(* PLC project copie_batch, Dassault Systèmes ControlBuild 2024x Refresh1 *)
(* stored: creationDateTime 2024-04-12T14:05:58-01:00 *)

PROGRAM gene_panel
  VAR_OUTPUT
    acknowledgePB : BOOL := false;
  END_VAR
  VAR_OUTPUT
    powerUp : BOOL := false;
    emergencyStop : BOOL := false;
    manualSwitch : BOOL := false;
    autoSwitch : BOOL := false;
    startCyclePB : BOOL := false;
    endCyclePB : BOOL := false;
  END_VAR

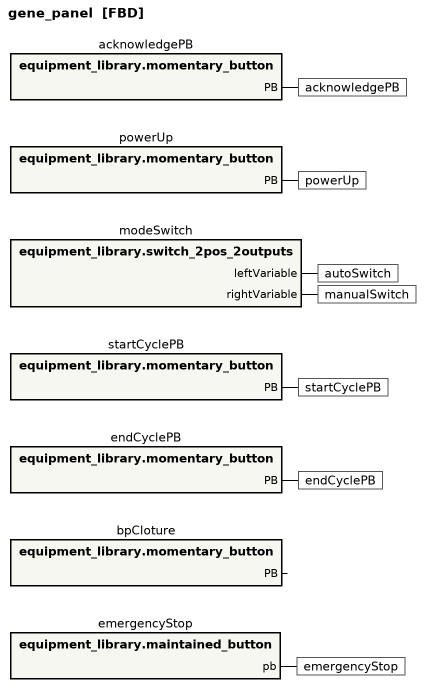
(* FBD diagram, written out as Structured Text *)
acknowledgePB();
acknowledgePB := acknowledgePB.PB;
powerUp();
powerUp := powerUp.PB;
emergencyStop();
emergencyStop := emergencyStop.pb;
modeSwitch();
autoSwitch := modeSwitch.leftVariable;
manualSwitch := modeSwitch.rightVariable;
startCyclePB();
startCyclePB := startCyclePB.PB;
endCyclePB();
endCyclePB := endCyclePB.PB;
bpCloture();
END_PROGRAM

PROGRAM copie_batch.copie_batch

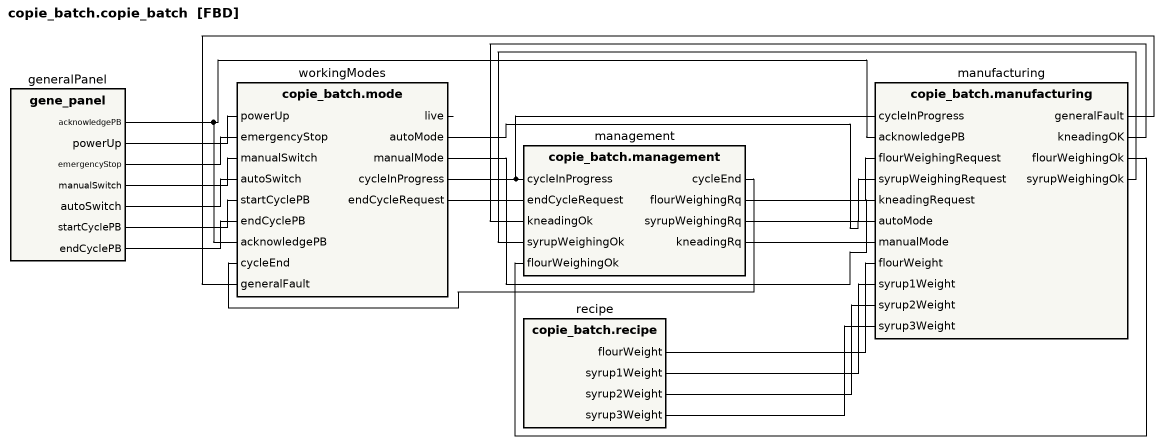
(* FBD diagram, written out as Structured Text *)
generalPanel();
management(cycleInProgress := workingModes.cycleInProgress, endCycleRequest := workingModes.endCycleRequest, kneadingOk := manufacturing.kneadingOK, syrupWeighingOk := manufacturing.syrupWeighingOk, flourWeighingOk := manufacturing.flourWeighingOk);
workingModes(powerUp := generalPanel.powerUp, emergencyStop := generalPanel.emergencyStop, manualSwitch := generalPanel.manualSwitch, autoSwitch := generalPanel.autoSwitch, startCyclePB := generalPanel.startCyclePB, endCyclePB := generalPanel.endCyclePB, acknowledgePB := generalPanel.acknowledgePB, cycleEnd := management.cycleEnd, generalFault := manufacturing.generalFault);
recipe();
manufacturing(cycleInProgress := workingModes.cycleInProgress, acknowledgePB := generalPanel.acknowledgePB, flourWeighingRequest := management.flourWeighingRq, syrupWeighingRequest := management.syrupWeighingRq, kneadingRequest := management.kneadingRq, autoMode := workingModes.autoMode, manualMode := workingModes.manualMode, flourWeight := recipe.flourWeight, syrup1Weight := recipe.syrup1Weight, syrup2Weight := recipe.syrup2Weight, syrup3Weight := recipe.syrup3Weight);
END_PROGRAM
